PROGRAM MAIN
VAR
	init_		:		init;
	handle1_	:		handle;
	clear_err_	:		clear_err;
	err_		:		err;
	reset_		:		reset;
	self_check_ :       SelfCheck;
	arm_manual_ :       ArmManual;
	axis2_sync_ :       Axis2Sync;
	injector_manual_ :  InjectorManual;
	axis6_enable_negative : BOOL := TRUE;
	i:INT;
END_VAR

FOR i:=1 TO 7 DO
	G.axis[i]();	
END_FOR

// 注射器 NC 轴刷新 AXIS_REF，由独立点动 POU 控制，不进入业务状态机。
FOR i:=1 TO 2 DO
	G.inject_axis[i]();
END_FOR

IF TwinCAT_SystemInfoVarList._TaskInfo[1].FirstCycle THEN
	G.gen_state := _init;
	G.self_check_done := FALSE;
	G.handle_reinit_req := FALSE;
	G.handle_reinit_done := FALSE;
	G.estop_hold_req := TRUE;
	G.selfcheck_reset_req := TRUE;
	FOR i:=1 TO 7 DO
		G.SetPointGenEnable[i].Execute := FALSE;
		G.SetPointGenDisable[i].Execute := FALSE;
		G.axis_Reset[i].Execute := FALSE;
	END_FOR
	G.arm_manual_enable := FALSE;
	FOR i:=1 TO 5 DO
		// PLC 启动时定位臂必须保持断使能，不能因为残留请求自动上电。
		G.arm_enable_req[i] := FALSE;
		G.arm_reset_req[i] := FALSE;
		G.arm_jog_pos_req[i] := FALSE;
		G.arm_jog_neg_req[i] := FALSE;
	END_FOR
END_IF
	
arm_manual_();
axis2_sync_();
injector_manual_();

// 轴6自检触发左限位后只关闭负向许可，保留正向脱离限位的能力。
axis6_enable_negative := NOT ((G.gen_state = _self_check) AND G.axis[6].Status.DriveLimitActive);
POWERED();
SETPOSITIONGEN();
RESETED();

CASE G.gen_state OF
	_init:			init_();
	_self_check:    self_check_();
	_handle:		handle1_();	
	_clear_err:		clear_err_();	
	_err:			err_();	
	_reset:			reset_();
END_CASE

ACTION POWERED:
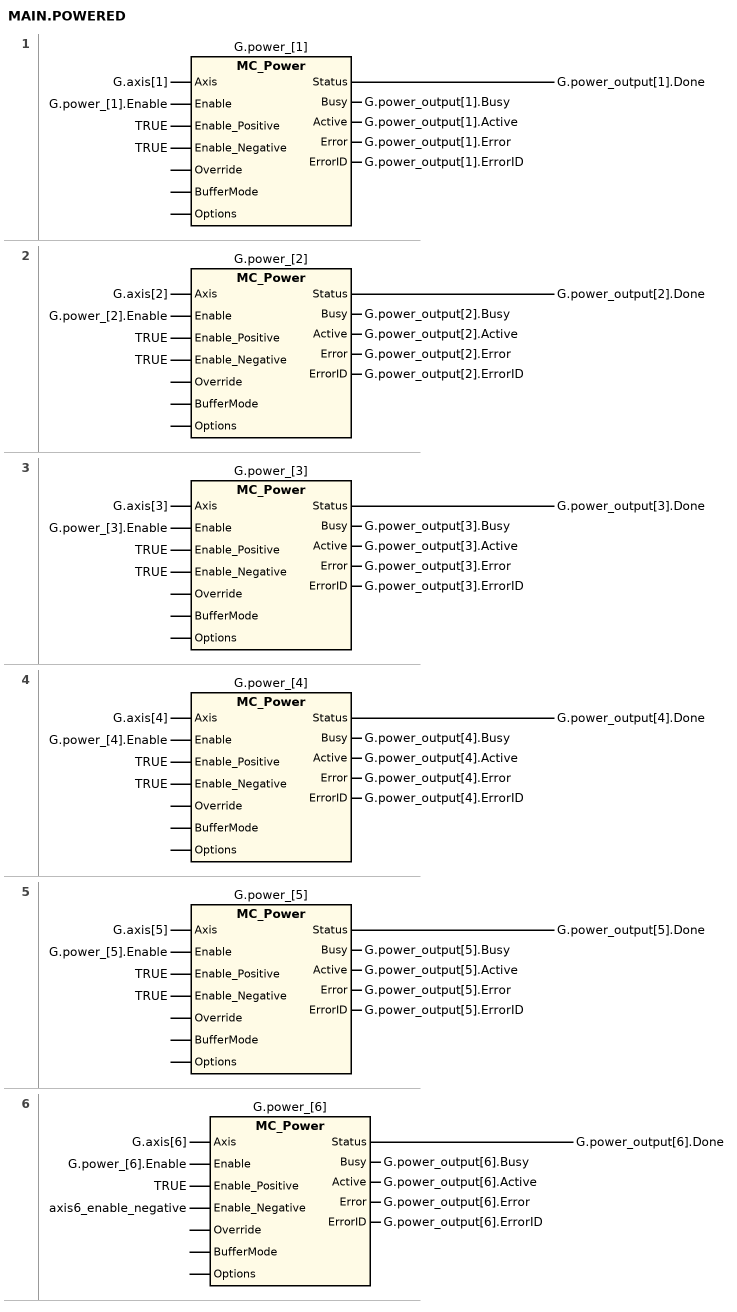
// NETWORK 1
G.power_[1](
    Axis := G.axis[1],
    Enable := G.power_[1].Enable,
    Enable_Positive := TRUE,
    Enable_Negative := TRUE,
    Busy => G.power_output[1].Busy,
    Active => G.power_output[1].Active,
    Error => G.power_output[1].Error,
    ErrorID => G.power_output[1].ErrorID); // MC_Power
G.power_output[1].Done := G.power_[1].Status;

// NETWORK 2
G.power_[2](
    Axis := G.axis[2],
    Enable := G.power_[2].Enable,
    Enable_Positive := TRUE,
    Enable_Negative := TRUE,
    Busy => G.power_output[2].Busy,
    Active => G.power_output[2].Active,
    Error => G.power_output[2].Error,
    ErrorID => G.power_output[2].ErrorID); // MC_Power
G.power_output[2].Done := G.power_[2].Status;

// NETWORK 3
G.power_[3](
    Axis := G.axis[3],
    Enable := G.power_[3].Enable,
    Enable_Positive := TRUE,
    Enable_Negative := TRUE,
    Busy => G.power_output[3].Busy,
    Active => G.power_output[3].Active,
    Error => G.power_output[3].Error,
    ErrorID => G.power_output[3].ErrorID); // MC_Power
G.power_output[3].Done := G.power_[3].Status;

// NETWORK 4
G.power_[4](
    Axis := G.axis[4],
    Enable := G.power_[4].Enable,
    Enable_Positive := TRUE,
    Enable_Negative := TRUE,
    Busy => G.power_output[4].Busy,
    Active => G.power_output[4].Active,
    Error => G.power_output[4].Error,
    ErrorID => G.power_output[4].ErrorID); // MC_Power
G.power_output[4].Done := G.power_[4].Status;

// NETWORK 5
G.power_[5](
    Axis := G.axis[5],
    Enable := G.power_[5].Enable,
    Enable_Positive := TRUE,
    Enable_Negative := TRUE,
    Busy => G.power_output[5].Busy,
    Active => G.power_output[5].Active,
    Error => G.power_output[5].Error,
    ErrorID => G.power_output[5].ErrorID); // MC_Power
G.power_output[5].Done := G.power_[5].Status;

// NETWORK 6
G.power_[6](
    Axis := G.axis[6],
    Enable := G.power_[6].Enable,
    Enable_Positive := TRUE,
    Enable_Negative := axis6_enable_negative,
    Busy => G.power_output[6].Busy,
    Active => G.power_output[6].Active,
    Error => G.power_output[6].Error,
    ErrorID => G.power_output[6].ErrorID); // MC_Power
G.power_output[6].Done := G.power_[6].Status;

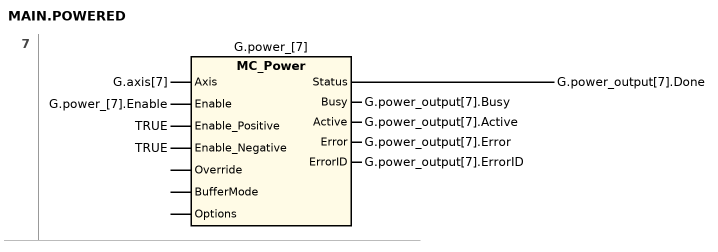
// NETWORK 7
G.power_[7](
    Axis := G.axis[7],
    Enable := G.power_[7].Enable,
    Enable_Positive := TRUE,
    Enable_Negative := TRUE,
    Busy => G.power_output[7].Busy,
    Active => G.power_output[7].Active,
    Error => G.power_output[7].Error,
    ErrorID => G.power_output[7].ErrorID); // MC_Power
G.power_output[7].Done := G.power_[7].Status;
END_ACTION

ACTION RESETED:
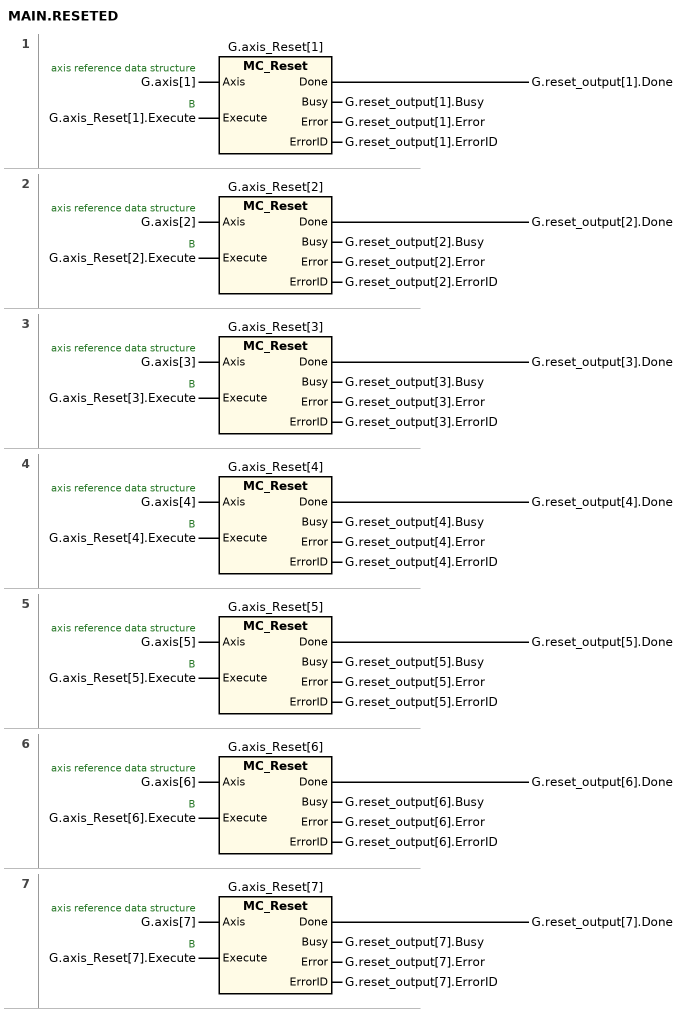
// NETWORK 1
//   G.axis[1]: axis reference data structure
//   G.axis_Reset[1].Execute: B
G.axis_Reset[1](
    Axis := G.axis[1],
    Execute := G.axis_Reset[1].Execute,
    Busy => G.reset_output[1].Busy,
    Error => G.reset_output[1].Error,
    ErrorID => G.reset_output[1].ErrorID); // MC_Reset
G.reset_output[1].Done := G.axis_Reset[1].Done;

// NETWORK 2
//   G.axis[2]: axis reference data structure
//   G.axis_Reset[2].Execute: B
G.axis_Reset[2](
    Axis := G.axis[2],
    Execute := G.axis_Reset[2].Execute,
    Busy => G.reset_output[2].Busy,
    Error => G.reset_output[2].Error,
    ErrorID => G.reset_output[2].ErrorID); // MC_Reset
G.reset_output[2].Done := G.axis_Reset[2].Done;

// NETWORK 3
//   G.axis[3]: axis reference data structure
//   G.axis_Reset[3].Execute: B
G.axis_Reset[3](
    Axis := G.axis[3],
    Execute := G.axis_Reset[3].Execute,
    Busy => G.reset_output[3].Busy,
    Error => G.reset_output[3].Error,
    ErrorID => G.reset_output[3].ErrorID); // MC_Reset
G.reset_output[3].Done := G.axis_Reset[3].Done;

// NETWORK 4
//   G.axis[4]: axis reference data structure
//   G.axis_Reset[4].Execute: B
G.axis_Reset[4](
    Axis := G.axis[4],
    Execute := G.axis_Reset[4].Execute,
    Busy => G.reset_output[4].Busy,
    Error => G.reset_output[4].Error,
    ErrorID => G.reset_output[4].ErrorID); // MC_Reset
G.reset_output[4].Done := G.axis_Reset[4].Done;

// NETWORK 5
//   G.axis[5]: axis reference data structure
//   G.axis_Reset[5].Execute: B
G.axis_Reset[5](
    Axis := G.axis[5],
    Execute := G.axis_Reset[5].Execute,
    Busy => G.reset_output[5].Busy,
    Error => G.reset_output[5].Error,
    ErrorID => G.reset_output[5].ErrorID); // MC_Reset
G.reset_output[5].Done := G.axis_Reset[5].Done;

// NETWORK 6
//   G.axis[6]: axis reference data structure
//   G.axis_Reset[6].Execute: B
G.axis_Reset[6](
    Axis := G.axis[6],
    Execute := G.axis_Reset[6].Execute,
    Busy => G.reset_output[6].Busy,
    Error => G.reset_output[6].Error,
    ErrorID => G.reset_output[6].ErrorID); // MC_Reset
G.reset_output[6].Done := G.axis_Reset[6].Done;

// NETWORK 7
//   G.axis[7]: axis reference data structure
//   G.axis_Reset[7].Execute: B
G.axis_Reset[7](
    Axis := G.axis[7],
    Execute := G.axis_Reset[7].Execute,
    Busy => G.reset_output[7].Busy,
    Error => G.reset_output[7].Error,
    ErrorID => G.reset_output[7].ErrorID); // MC_Reset
G.reset_output[7].Done := G.axis_Reset[7].Done;
END_ACTION

ACTION SETPOSITIONGEN:
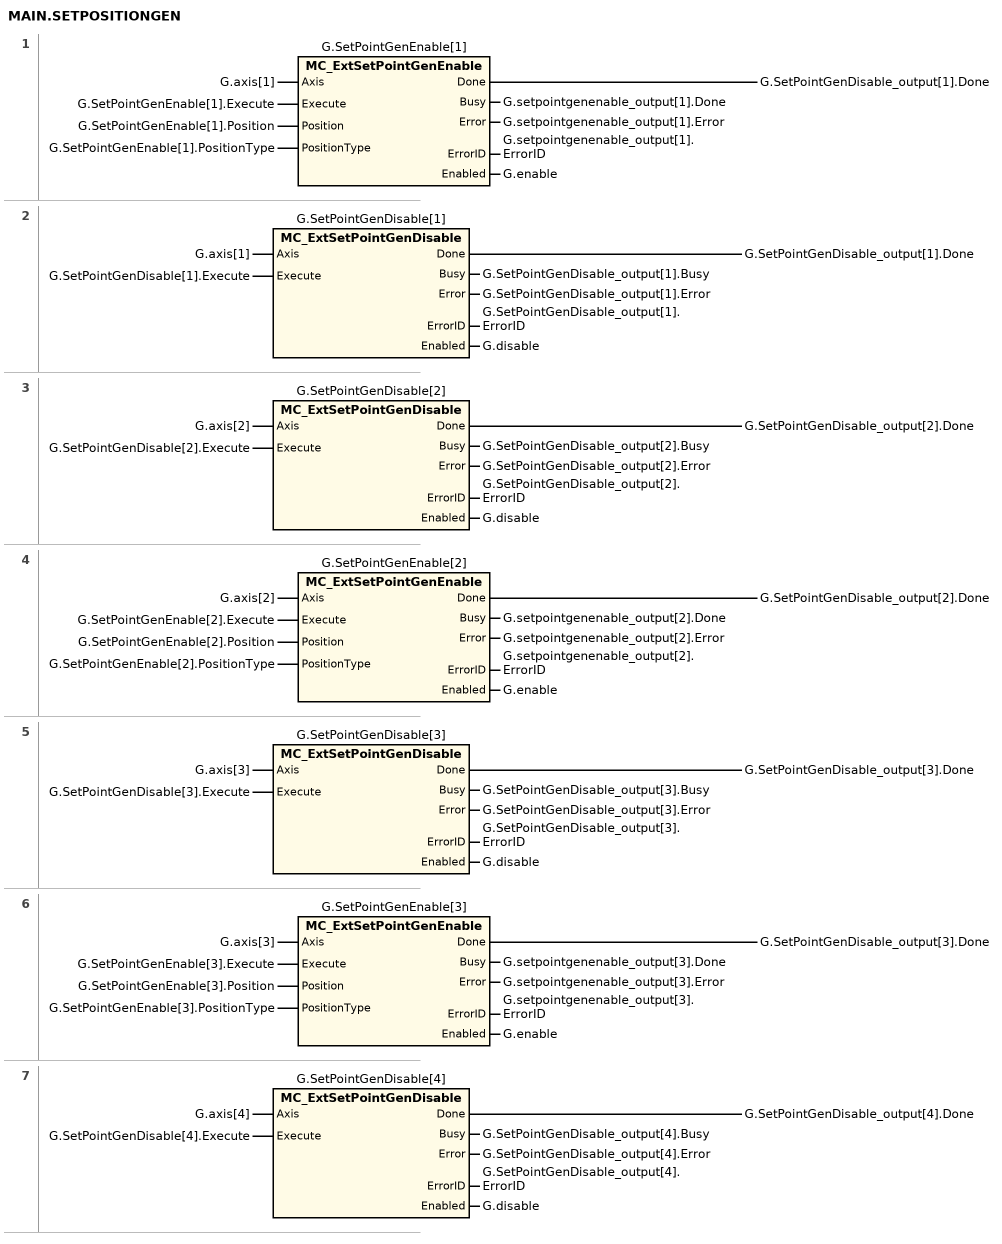
// NETWORK 1
G.SetPointGenEnable[1](
    Axis := G.axis[1],
    Execute := G.SetPointGenEnable[1].Execute,
    Position := G.SetPointGenEnable[1].Position,
    PositionType := G.SetPointGenEnable[1].PositionType,
    Busy => G.setpointgenenable_output[1].Done,
    Error => G.setpointgenenable_output[1].Error,
    ErrorID => G.setpointgenenable_output[1].ErrorID,
    Enabled => G.enable); // MC_ExtSetPointGenEnable
G.SetPointGenDisable_output[1].Done := G.SetPointGenEnable[1].Done;

// NETWORK 2
G.SetPointGenDisable[1](
    Axis := G.axis[1],
    Execute := G.SetPointGenDisable[1].Execute,
    Busy => G.SetPointGenDisable_output[1].Busy,
    Error => G.SetPointGenDisable_output[1].Error,
    ErrorID => G.SetPointGenDisable_output[1].ErrorID,
    Enabled => G.disable); // MC_ExtSetPointGenDisable
G.SetPointGenDisable_output[1].Done := G.SetPointGenDisable[1].Done;

// NETWORK 3
G.SetPointGenDisable[2](
    Axis := G.axis[2],
    Execute := G.SetPointGenDisable[2].Execute,
    Busy => G.SetPointGenDisable_output[2].Busy,
    Error => G.SetPointGenDisable_output[2].Error,
    ErrorID => G.SetPointGenDisable_output[2].ErrorID,
    Enabled => G.disable); // MC_ExtSetPointGenDisable
G.SetPointGenDisable_output[2].Done := G.SetPointGenDisable[2].Done;

// NETWORK 4
G.SetPointGenEnable[2](
    Axis := G.axis[2],
    Execute := G.SetPointGenEnable[2].Execute,
    Position := G.SetPointGenEnable[2].Position,
    PositionType := G.SetPointGenEnable[2].PositionType,
    Busy => G.setpointgenenable_output[2].Done,
    Error => G.setpointgenenable_output[2].Error,
    ErrorID => G.setpointgenenable_output[2].ErrorID,
    Enabled => G.enable); // MC_ExtSetPointGenEnable
G.SetPointGenDisable_output[2].Done := G.SetPointGenEnable[2].Done;

// NETWORK 5
G.SetPointGenDisable[3](
    Axis := G.axis[3],
    Execute := G.SetPointGenDisable[3].Execute,
    Busy => G.SetPointGenDisable_output[3].Busy,
    Error => G.SetPointGenDisable_output[3].Error,
    ErrorID => G.SetPointGenDisable_output[3].ErrorID,
    Enabled => G.disable); // MC_ExtSetPointGenDisable
G.SetPointGenDisable_output[3].Done := G.SetPointGenDisable[3].Done;

// NETWORK 6
G.SetPointGenEnable[3](
    Axis := G.axis[3],
    Execute := G.SetPointGenEnable[3].Execute,
    Position := G.SetPointGenEnable[3].Position,
    PositionType := G.SetPointGenEnable[3].PositionType,
    Busy => G.setpointgenenable_output[3].Done,
    Error => G.setpointgenenable_output[3].Error,
    ErrorID => G.setpointgenenable_output[3].ErrorID,
    Enabled => G.enable); // MC_ExtSetPointGenEnable
G.SetPointGenDisable_output[3].Done := G.SetPointGenEnable[3].Done;

// NETWORK 7
G.SetPointGenDisable[4](
    Axis := G.axis[4],
    Execute := G.SetPointGenDisable[4].Execute,
    Busy => G.SetPointGenDisable_output[4].Busy,
    Error => G.SetPointGenDisable_output[4].Error,
    ErrorID => G.SetPointGenDisable_output[4].ErrorID,
    Enabled => G.disable); // MC_ExtSetPointGenDisable
G.SetPointGenDisable_output[4].Done := G.SetPointGenDisable[4].Done;

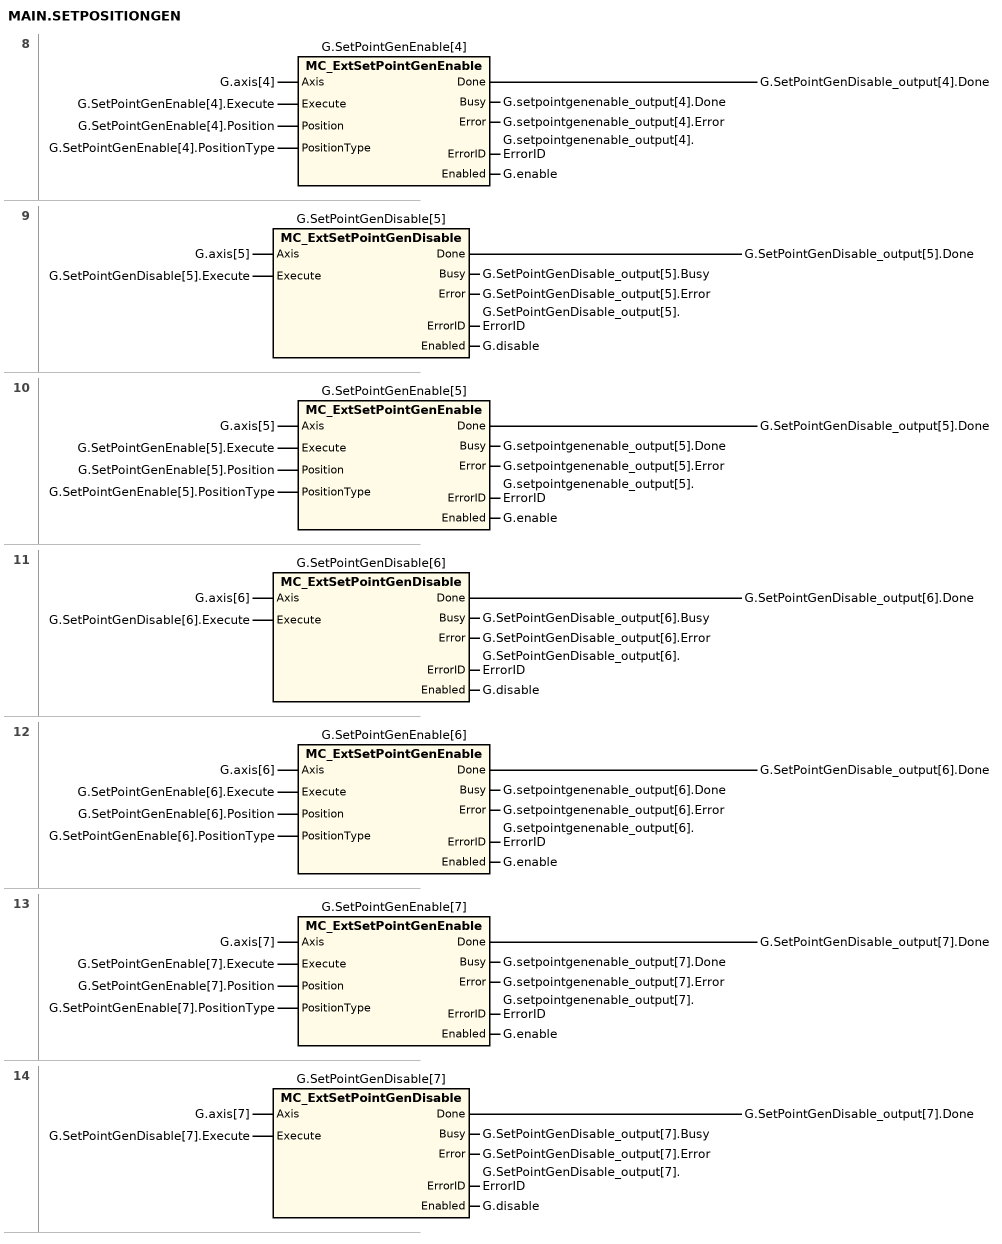
// NETWORK 8
G.SetPointGenEnable[4](
    Axis := G.axis[4],
    Execute := G.SetPointGenEnable[4].Execute,
    Position := G.SetPointGenEnable[4].Position,
    PositionType := G.SetPointGenEnable[4].PositionType,
    Busy => G.setpointgenenable_output[4].Done,
    Error => G.setpointgenenable_output[4].Error,
    ErrorID => G.setpointgenenable_output[4].ErrorID,
    Enabled => G.enable); // MC_ExtSetPointGenEnable
G.SetPointGenDisable_output[4].Done := G.SetPointGenEnable[4].Done;

// NETWORK 9
G.SetPointGenDisable[5](
    Axis := G.axis[5],
    Execute := G.SetPointGenDisable[5].Execute,
    Busy => G.SetPointGenDisable_output[5].Busy,
    Error => G.SetPointGenDisable_output[5].Error,
    ErrorID => G.SetPointGenDisable_output[5].ErrorID,
    Enabled => G.disable); // MC_ExtSetPointGenDisable
G.SetPointGenDisable_output[5].Done := G.SetPointGenDisable[5].Done;

// NETWORK 10
G.SetPointGenEnable[5](
    Axis := G.axis[5],
    Execute := G.SetPointGenEnable[5].Execute,
    Position := G.SetPointGenEnable[5].Position,
    PositionType := G.SetPointGenEnable[5].PositionType,
    Busy => G.setpointgenenable_output[5].Done,
    Error => G.setpointgenenable_output[5].Error,
    ErrorID => G.setpointgenenable_output[5].ErrorID,
    Enabled => G.enable); // MC_ExtSetPointGenEnable
G.SetPointGenDisable_output[5].Done := G.SetPointGenEnable[5].Done;

// NETWORK 11
G.SetPointGenDisable[6](
    Axis := G.axis[6],
    Execute := G.SetPointGenDisable[6].Execute,
    Busy => G.SetPointGenDisable_output[6].Busy,
    Error => G.SetPointGenDisable_output[6].Error,
    ErrorID => G.SetPointGenDisable_output[6].ErrorID,
    Enabled => G.disable); // MC_ExtSetPointGenDisable
G.SetPointGenDisable_output[6].Done := G.SetPointGenDisable[6].Done;

// NETWORK 12
G.SetPointGenEnable[6](
    Axis := G.axis[6],
    Execute := G.SetPointGenEnable[6].Execute,
    Position := G.SetPointGenEnable[6].Position,
    PositionType := G.SetPointGenEnable[6].PositionType,
    Busy => G.setpointgenenable_output[6].Done,
    Error => G.setpointgenenable_output[6].Error,
    ErrorID => G.setpointgenenable_output[6].ErrorID,
    Enabled => G.enable); // MC_ExtSetPointGenEnable
G.SetPointGenDisable_output[6].Done := G.SetPointGenEnable[6].Done;

// NETWORK 13
G.SetPointGenEnable[7](
    Axis := G.axis[7],
    Execute := G.SetPointGenEnable[7].Execute,
    Position := G.SetPointGenEnable[7].Position,
    PositionType := G.SetPointGenEnable[7].PositionType,
    Busy => G.setpointgenenable_output[7].Done,
    Error => G.setpointgenenable_output[7].Error,
    ErrorID => G.setpointgenenable_output[7].ErrorID,
    Enabled => G.enable); // MC_ExtSetPointGenEnable
G.SetPointGenDisable_output[7].Done := G.SetPointGenEnable[7].Done;

// NETWORK 14
G.SetPointGenDisable[7](
    Axis := G.axis[7],
    Execute := G.SetPointGenDisable[7].Execute,
    Busy => G.SetPointGenDisable_output[7].Busy,
    Error => G.SetPointGenDisable_output[7].Error,
    ErrorID => G.SetPointGenDisable_output[7].ErrorID,
    Enabled => G.disable); // MC_ExtSetPointGenDisable
G.SetPointGenDisable_output[7].Done := G.SetPointGenDisable[7].Done;
END_ACTION

END_PROGRAM

(* stored: Version 1.1.0.1, ProductVersion 3.1.4024.15
   POU MAIN: Id {0f7d3262-e451-4dc7-838c-99daae61b3ae}, SpecialFunc None
   Folder block: Id {8d2a06f7-1a45-482f-85f8-8678060c15b3}
   Action POWERED: Id {98a6d293-ca3a-4d71-85c7-080c2df57892}
   Action RESETED: Id {8998d5fe-e5f4-45d3-81ca-7f0717ea31dd}
   Action SETPOSITIONGEN: Id {37f9e6a4-cc02-4cfa-997f-805ef02e2982} *)
